{attribute 'linkalways'} 
{attribute 'no_explicit_call' := 'This FB is a CLASS and must be accessed using methods or properties'}
{attribute 'enable_dynamic_creation'}
FUNCTION_BLOCK _TcVnParamsBRISK EXTENDS StructuredDatatypeBase
VAR
	localData : TcVnParamsBRISK;
	activeData : REFERENCE TO TcVnParamsBRISK REF= localData;
	_nThreshold : _DINT(localData.nThreshold);
	_nOctaves : _UDINT(localData.nOctaves);
	_fPatternScale : _REAL(localData.fPatternScale);
END_VAR

PROPERTY PUBLIC Address : PVOID
GET
Address := ADR(activeData);
END_GET
END_PROPERTY

METHOD PUBLIC ClearReference
VAR_INPUT
END_VAR
activeData REF= localData;
SetMemberReference();
END_METHOD

METHOD PUBLIC Clone : I_Datatype
VAR
    pClone : POINTER TO _TcVnParamsBRISK;
END_VAR
pClone := __NEW(_TcVnParamsBRISK());
pClone^.Value := Value;
Clone := pClone^;
END_METHOD

METHOD FB_init : BOOL
VAR_INPUT
	bInitRetains : BOOL; // if TRUE, the retain variables are initialized (warm start / cold start)
	bInCopyCode : BOOL;  // if TRUE, the instance afterwards gets moved into the copy code (online change)
END_VAR
SetMemberReference();
AddMember('nThreshold', _nThreshold);
AddMember('nOctaves', _nOctaves);
AddMember('fPatternScale', _fPatternScale);
END_METHOD

PROPERTY PUBLIC fPatternScale : REFERENCE TO _REAL
GET
fPatternScale REF= _fPatternScale;
END_GET
END_PROPERTY

PROPERTY PUBLIC Identifier : T_MAXSTRING
GET
Identifier := 'TcVnParamsBRISK';
END_GET
END_PROPERTY

METHOD PUBLIC MakeReferenceTo
VAR_INPUT
	ReferenceTarget : REFERENCE TO TcVnParamsBRISK;
END_VAR
activeData REF= ReferenceTarget;
SetMemberReference();
END_METHOD

PROPERTY PUBLIC nOctaves : REFERENCE TO _UDINT
GET
nOctaves REF= _nOctaves;
END_GET
END_PROPERTY

PROPERTY PUBLIC nThreshold : REFERENCE TO _DINT
GET
nThreshold REF= _nThreshold;
END_GET
END_PROPERTY

METHOD PROTECTED SetMemberReference
VAR_INPUT
END_VAR
_nThreshold.MakeReferenceTo(activeData.nThreshold);
_nOctaves.MakeReferenceTo(activeData.nOctaves);
_fPatternScale.MakeReferenceTo(activeData.fPatternScale);
END_METHOD

PROPERTY PUBLIC Size : UDINT
GET
Size := SIZEOF(activeData);
END_GET
END_PROPERTY

METHOD TryMakeReferenceTo : BOOL
VAR_INPUT
	Target : I_Datatype;
END_VAR
VAR
	pTargetData : POINTER TO TcVnParamsBRISK;
END_VAR
IF NOT IsEquivalentTo(Target) THEN
	RETURN;
END_IF

pTargetData := Target.Address;
activeData REF= pTargetData^;
SetMemberReference();
TryMakeReferenceTo := TRUE;
END_METHOD

PROPERTY PUBLIC Value : REFERENCE TO TcVnParamsBRISK
GET
Value REF= activeData;
END_GET
END_PROPERTY

METHOD PUBLIC TryDeserializeFrom : BOOL
VAR_INPUT
    Deserializer : I_Deserializer;
    Feedback : I_DeserializerFeedback;
END_VAR
VAR
    membersEnumerator : I_DeserializerObjectForwardEnumerator;
    member : I_Datatype;
    memberName : T_MAXSTRING;
END_VAR
// Map the legacy member name without advertising or serializing it twice.
membersEnumerator := Deserializer.GetObjectEnumerator();
WHILE membersEnumerator.MoveNext() DO
    memberName := membersEnumerator.Key;
    IF memberName = 'fPatternScale ' THEN
        memberName := 'fPatternScale';
    END_IF
    IF Members.TryGetMemberByName(memberName, member) THEN
        IF NOT member.TryDeserializeFrom(membersEnumerator.Current, Feedback) THEN
            membersEnumerator.Dispose();
            RETURN;
        END_IF
    END_IF
END_WHILE
membersEnumerator.Dispose();
TryDeserializeFrom := TRUE;
END_METHOD

END_FUNCTION_BLOCK

(* stored: Version 1.1.0.1, ProductVersion 3.1.4024.13
   POU _TcVnParamsBRISK: Id {3fcecca7-1e19-0428-333d-fd893c5d7297}, SpecialFunc None
   Folder Core: Id {2cbea202-f2fb-039b-2c1f-acca9683f1a5}
   Folder Customize: Id {3d6b6e48-7866-08d3-1d83-17cbc67de8b9}
   Folder Constructor: Id {b1a1d65a-6a88-09fe-3aed-093a04e97340}
   Folder Protected: Id {828001e8-2b47-0ebb-349d-8f4efda51371}
   Property Address: Id {1c3b9f53-ebc2-0070-374f-c065c67f97c9}
   Get Get: Id {2b01aa63-5513-0cba-17e2-32480a5988c4}
   Method ClearReference: Id {5d47f96b-244e-0fc9-25e6-d407bb02559e}
   Method Clone: Id {078e0be9-13aa-05d5-2bde-7a0928995e08}
   Method FB_init: Id {6d734615-bae3-061c-1191-743e4766c09f}
   Property fPatternScale: Id {78f5b869-8edb-0ec3-20ef-5c8f9b9ce0e3}
   Get Get: Id {2c6fcb79-36d4-0b3d-2a22-98c389e22f68}
   Property Identifier: Id {ecf99577-2612-081f-0438-c7ed1997bbcb}
   Get Get: Id {af837c1e-b48a-0506-20f6-04560b901286}
   Method MakeReferenceTo: Id {1fec4d4a-e2b8-0b98-21b3-1c23d0bc378e}
   Property nOctaves: Id {b7105735-295f-0f47-0cb8-dad7161abac0}
   Get Get: Id {aab5ad4d-2d19-0cc1-0dfc-de8fd7a3415d}
   Property nThreshold: Id {0282dc74-5a63-02c7-3bf9-a4274c0a1108}
   Get Get: Id {74cfa11a-0e95-0088-01b7-dd2a1a2172d0}
   Method SetMemberReference: Id {6bfe8884-d1a1-0c57-3ccb-e8c9da37e45c}
   Property Size: Id {c5773d88-ebeb-090c-310a-ee5bde781632}
   Get Get: Id {67f9b54e-27ee-0158-23f8-008cdf5fbe12}
   Method TryMakeReferenceTo: Id {1b481c9e-b7e3-0ddc-162c-548f95f216af}
   Property Value: Id {fe8c64d2-f3af-0599-240e-35da031c660f}
   Get Get: Id {00e1192c-899b-00c2-3274-129d06bf599c}
   Method TryDeserializeFrom: Id {3beb9d15-b8f7-49f1-b9d0-b17ee0db4796} *)
